{attribute 'linkalways'} 
{attribute 'no_explicit_call' := 'This FB is a CLASS and must be accessed using methods or properties'}
{attribute 'enable_dynamic_creation'}
FUNCTION_BLOCK BasicNodePack IMPLEMENTS I_NodePack
VAR
	booleanLiteralNode : BooleanLiteralNode;
	booleanDisplayNode : BooleanDisplayNode;
	intLiteralNode : IntLiteralNode;
	intDisplayNode : IntDisplayNode;
	realLiteralNode : RealLiteralNode;
	realDisplayNode : RealDisplayNode;
END_VAR

METHOD PUBLIC RegisterWithNodeFactory
VAR_INPUT
	NodeFactory : I_NodeFactory;
END_VAR
NodeFactory.AddNodeAsPrototype('PlcBasic.Bool.BoolLiteral',booleanLiteralNode);
NodeFactory.AddNodeAsPrototype('PlcBasic.Bool.BoolDisplay',booleanDisplayNode);
NodeFactory.AddNodeAsPrototype('PlcBasic.Int.IntLiteral',intLiteralNode);
NodeFactory.AddNodeAsPrototype('PlcBasic.Int.IntDisplay',intDisplayNode);
NodeFactory.AddNodeAsPrototype('PlcBasic.Real.RealLiteral',realLiteralNode);
NodeFactory.AddNodeAsPrototype('PlcBasic.Real.RealDisplay',realDisplayNode);
END_METHOD

END_FUNCTION_BLOCK

(* stored: Version 1.1.0.1, ProductVersion 3.1.4024.12
   POU BasicNodePack: Id {764b13ce-dfc8-0116-1a3e-aea066c68a36}, SpecialFunc None
   Method RegisterWithNodeFactory: Id {cdeee486-eac2-0e76-1902-0e4879666445} *)
